Staubli VAL3: HerePointCircle.pgx

public program HerePointCircle(num x_nIndex)
  local tool l_tTool
  local point l_pHere
  local frame l_fFrame
  local num i
  local num l_nIndex
  local num l_nSize
begin
  //
  // take the point
  //
  // frame
  call getFrame(fSetFrame,false)
  // tool
  call tcp:getTool(l_tTool,pEditPoint.nIndexTool)
  // here
  l_pHere=here(l_tTool,fSetFrame)
  resetMotion()
  // save the trsf
  pEditPoint.tData[x_nIndex].pCircle.trsf=l_pHere.trsf
  // check the moveType to save the config
  if pEditPoint.tData[x_nIndex].tSuper.moveType==0
    pEditPoint.tData[x_nIndex].pCircle.config=l_pHere.config
  endIf
end
